TYPE ENCStatusCompactChannel :
STRUCT
	{attribute addProperty Name "Status"}
	Status AT %I* : stENCStatusCompact;
	{attribute addProperty Name "Counter value"}
	CounterValue AT %I* : UINT;
END_STRUCT
END_TYPE

(* stored: Version 1.1.0.1, ProductVersion 3.1.4024.9
   DUT ENCStatusCompactChannel: Id {88b5c7b2-368a-06b0-31b4-f3658569d5f9} *)
